TYPE ST_AxisSettings :
STRUCT
	MovePosAcc : LREAL;
	MovePosDec : LREAL;
	MovePosJerk : LREAL;
	
	MoveVeloAcc : LREAL;
	MoveVeloDec : LREAL;
	MoveVeloJerk : LREAL;
	MoveVeloDirection : MC_Direction := MC_Positive_Direction;
	
	JogAcc : LREAL;
	JogDec : LREAL;
	JogJerk : LREAL;
	
	HomeVelo : LREAL := 10;
	HomeAcc : LREAL;
	HomeDec : LREAL;
	HomeJerk : LREAL;
	HomeSetpos : LREAL := 0;
	HomeSignal : BOOL;
	HomePosLimit : BOOL;
	HomeNegLimit : BOOL;
END_STRUCT
END_TYPE

(* stored: Version 1.1.0.1, ProductVersion 3.1.4024.12
   DUT ST_AxisSettings: Id {37889c6e-6c9a-4f04-86db-bcfb836e22bc} *)
